{attribute 'GeneratedUsingTerminal: EK1122-0000-0018'}
{attribute addProperty BoxType "EK1122-0000-0018"}
{attribute addProperty Id "Beckhoff_EL34xxsub_EK1100EK1100_AB5A94672"}
{attribute addProperty CRC "1367866986"}
{attribute addProperty Size "2"}
TYPE Beckhoff_EL34xxEK1122_5187FE6A EXTENDS EK1122_AB5A9467 :
STRUCT
	{attribute addProperty Name "Beckhoff_EL34xxsub_EK1100"}
	{attribute addProperty PreviousPort "Beckhoff EL34xxEK1122 : D"}
	Beckhoff_EL34xxsub_EK1100 : EK1100_AB5A9467;
END_STRUCT
END_TYPE

(* stored: Version 1.2.0.0, ProductVersion 3.1.4024.9
   DUT Beckhoff_EL34xxEK1122_5187FE6A: Id {a170577b-aa3b-4681-bdfd-774c05020b37} *)
